// TwinCAT 3 PLC project ReceipeManager
// ProgramVersion: 3.1.4026.24
// libraries:
//   Tc2_Standard, * (Beckhoff Automation GmbH)
//   Tc2_System, * (Beckhoff Automation GmbH)
// project tree:
//   / PlcTask.TcTTO (not stored)
//   POUs/ MAIN.TcPOU (not stored)
//   GVLs/ GVL_Command.TcGVL, GVL_State.TcGVL (not stored), GVL_Recipe.TcGVL, GVL_Process.TcGVL

// ---- GVLs/GVL_Command.TcGVL
{attribute 'qualified_only'}
VAR_GLOBAL
    // PackML commands - written by the Blazor client as momentary pulses (TRUE then FALSE)
    bReset      : BOOL;
    bClear      : BOOL;
    bStart      : BOOL;
    bHold       : BOOL;
    bStop       : BOOL;

    // Set by the Blazor client right after a successful ADS connection
    bAdsConnected : BOOL;
END_VAR

// ---- GVLs/GVL_Recipe.TcGVL
{attribute 'qualified_only'}
VAR_GLOBAL CONSTANT
    MAX_STEPS       : UINT := 20;
    MAX_INGREDIENTS : UINT := 10;
END_VAR

VAR_GLOBAL
    // Recipe metadata - written by the Blazor client before Start
    sRecipeName             : STRING(254);
    fPreparationVolume      : REAL;
    fPreparationConcentration : REAL;

    // Ordered process step sequence (e.g. Dosage, Melange, Extraction, Cuisson)
    nNumSteps               : UINT;
    aStepNames              : ARRAY[1..20] OF STRING(254);

    // Ingredients and their quantities
    nNumIngredients         : UINT;
    aIngredientName         : ARRAY[1..10] OF STRING(254);
    aIngredientQuantity     : ARRAY[1..10] OF REAL;
    aIngredientVolume       : ARRAY[1..10] OF REAL;
    aIngredientMolarMass    : ARRAY[1..10] OF REAL;
END_VAR

// ---- GVLs/GVL_Process.TcGVL
{attribute 'qualified_only'}
VAR_GLOBAL
    // Live execution status - updated every PLC cycle, read by the Blazor client
    nCurrentStepIndex     : UINT;              // 1-based index into GVL_Recipe.aStepNames, 0 = none active
    sCurrentStepName      : STRING(254);
    nStepTimeElapsed_s    : UINT;               // 0..15
    nStepTimeRemaining_s  : UINT;               // 15..0
    nTotalSteps           : UINT;
    fProgress             : REAL;               // overall recipe progress 0.0..1.0
    bProcessDone          : BOOL;               // TRUE once state = Complete

    nErrorCode            : INT;
    sErrorText            : STRING(254);
END_VAR
